TYPE MoverSequenceInfo :
STRUCT
	MoverId : UDINT;
	CurrentStation : INT;
	Velocity : MC_LREAL;
	State : IndexSequenceState;
END_STRUCT
END_TYPE

(* stored: Version 1.1.0.1, ProductVersion 3.1.4024.11
   DUT MoverSequenceInfo: Id {e076e401-8b1f-40c9-8216-2b6b2d9b9748} *)
